FUNCTION_BLOCK FB_Button_Test EXTENDS TcUnit.FB_TestSuite
VAR
	fbButton : FB_Button;
	nExpected : BYTE;
	nResult : BYTE;
	bExpected : BOOL;
	bResult : BOOL;
END_VAR

TEST('Set bEnable TRUE');			 
fbButton.bEnable := TRUE; 
fbButton();
nExpected := 1;
nResult := fbButton.GetControl();
AssertEquals(Expected := nExpected,
             Actual := nResult,
             Message := 'Control value is not correct');	 
TEST_FINISHED();

TEST('Set bEnable FALSE');			 
fbButton.bEnable := FALSE; 
fbButton();
nExpected := 0;
nResult := fbButton.GetControl();
AssertEquals(Expected := nExpected,
             Actual := nResult,
             Message := 'Control value is not correct');	 
TEST_FINISHED();


TEST('Get bValue FALSE');
fbButton.SetStatus(0);
fbButton();
bExpected := FALSE;
bResult := fbButton.bValue;

AssertEquals(Expected := bExpected,
             Actual := bResult,
             Message := 'Value is not correct');	
TEST_FINISHED();

TEST('Get bValue TRUE');	
fbButton.SetStatus(1);
fbButton();
bExpected := 1;
bResult := fbButton.bValue;
AssertEquals(Expected := bExpected,
             Actual := bResult,
             Message := 'Control value is not correct');	 
TEST_FINISHED();

END_FUNCTION_BLOCK

(* stored: Version 1.1.0.1, ProductVersion 3.1.4024.12
   POU FB_Button_Test: Id {1d01b343-9218-07c7-1af2-fff3bf9f86c7}, SpecialFunc None *)
